{attribute 'GeneratedUsingTerminal: EJ2918-0000-0017'}
{attribute addProperty BoxType "EJ2918-0000-0017"}
{attribute addProperty Id "EtcSlaveTerminalBaseModule_1_FSOEModule_1_FSOE_7F12D29222Module_2_FSOUTModule_2_FSOUT_9813A38E8Module_3_DEVICEIOModule_3_DEVICEIO_5FA6B4E72Module_4_FSLOGICModule_4_FSLOGIC_DEAB45222WcStateAT %I*WcState_B516A2644InfoDataAT %I*InfoData_32EB74EA10"}
{attribute addProperty CRC "3339326943"}
{attribute addProperty Size "48"}
TYPE EJ2918_C70A15DF EXTENDS EtcSlaveTerminalBase :
STRUCT
	{attribute addProperty Name "Module_1_FSOE"}
	Module_1_FSOE : Module_1_FSOE_7F12D292;
	{attribute addProperty Name "Module_2_FSOUT"}
	Module_2_FSOUT : Module_2_FSOUT_9813A38E;
	{attribute addProperty Name "Module_3_DEVICEIO"}
	Module_3_DEVICEIO : Module_3_DEVICEIO_5FA6B4E7;
	{attribute addProperty Name "Module_4_FSLOGIC"}
	Module_4_FSLOGIC : Module_4_FSLOGIC_DEAB4522;
	{attribute addProperty Name "WcState"}
	WcState : WcState_B516A264;
	{attribute addProperty Name "InfoData"}
	InfoData : InfoData_32EB74EA;
END_STRUCT
END_TYPE

(* stored: Version 1.2.0.0, ProductVersion 3.1.4024.9
   DUT EJ2918_C70A15DF: Id {4f285987-f311-4d80-abf4-37cb42d854e7} *)
